ABB RobotStudio station: WriteNameStation.rspag

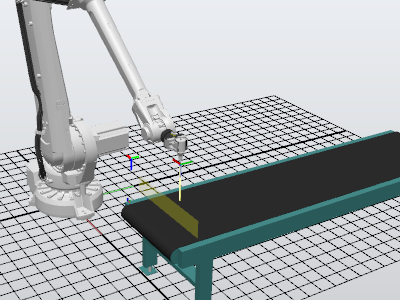
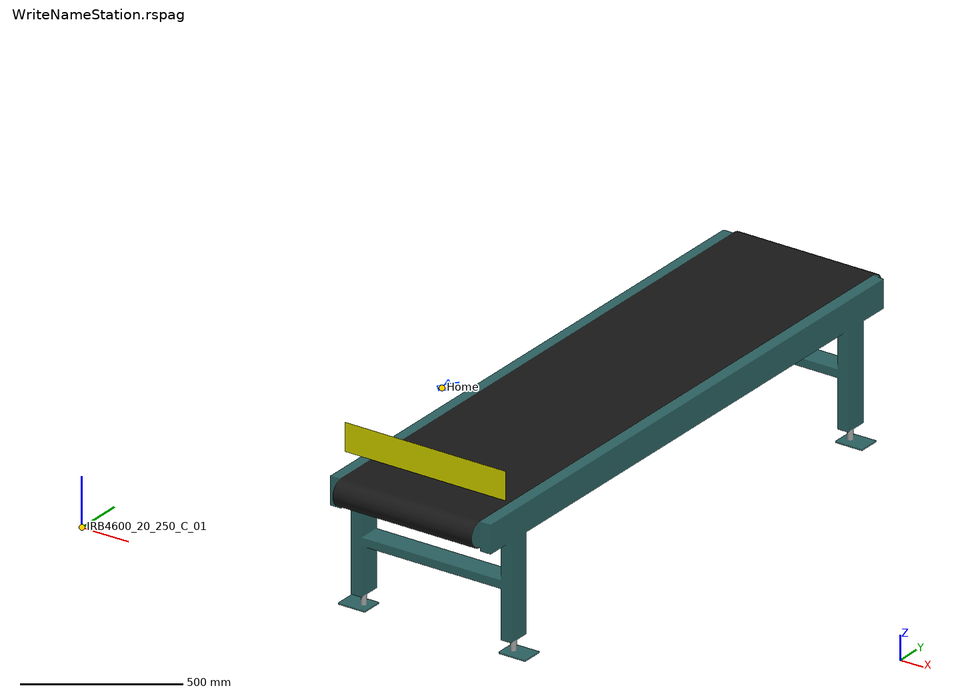
[picture v1: parts stored in the station drawn from their meshes, with robot base, taught points and paths (robot models come from the ABB library and are not in the file)]
--- station ---
Station WriteNameStation (saved by RobotStudio 23.4.10609.1)
Controller IRB4600
  mechanical unit ROB_1: IRB4600_20_250_C_01, 6 joints, base frame (0, 0, 0) mm
Layout (positions relative to the parent item):
  - IRB4600_20_250_C_01 [mechanism, from %ABB.RobotStudio.Models.IRB4600%\IRB4600_20_250_C_G_01.rslib] at (0, 0, 0) mm; joint values [0.065, -0.1396, 0.8384, 0.1009, -0.7014, -0.0772] (rad or m)
  - Belt Conveyor [part], size 703.5 x 2188.6 x 501 mm
  - Box [part], size 500 x 300 x 200 mm
  - SC_InFeeder [smart component]
      signals: DO doBoxInPos, DO doConveyorPaused, DI alwaysOn, DI diConveyor
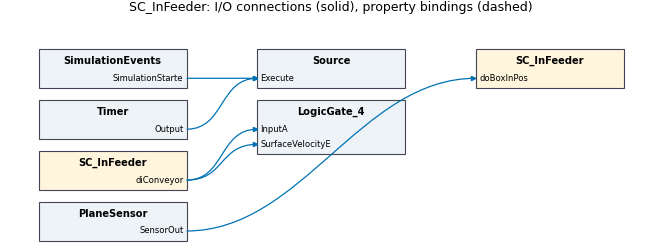
      connections:
        SimulationEvents.SimulationStarted -> Source.Execute
        Timer.Output -> Source.Execute
        SC_InFeeder.diConveyor -> LogicGate_4.InputA
        SC_InFeeder.diConveyor -> PhysicsControl.SurfaceVelocityEnabled
        PlaneSensor.SensorOut -> SC_InFeeder.doBoxInPos
    - Source [smart component, from Components\Source.rslib]
        properties: Source=Box; Copy=(none); Parent=(none); Position=[0 0 0]; Orientation=[0 0 0]; Transient=true; PhysicsBehavior=3
    - SimulationEvents [smart component, from Components\SimulationEvents.rslib]
    - Timer [smart component, from Components\Timer.rslib]
        properties: StartTime=0; Interval=5; Repeat=true; CurrentTime=12.288
    - PlaneSensor [smart component, from Components\PlaneSensor.rslib] at (984.64, 0, 535.74) mm, rotated rx 90 ry 0 rz 0 deg
        properties: Origin=[0 0 0]; Axis1=[0.6 0 0]; Axis2=[0 0.1 0]; Tag=(none); SensedPart=(none)
      - _sensorPart_ [part], size 600 x 100 x 0 mm
  - Belt [part], size 529.1 x 2200.3 x 102.1 mm
  - Pen [mechanism, from Training Objects\Pen.rslib] at (1160.02, 70, 921.71) mm, rotated rx 0 ry 90 rz 0 deg
  - SC_Painter [smart component] at (1300.02, 70, 811.71) mm, rotated rx 0 ry 0 rz -180 deg
      signals: DI diPaint
      connections:
        SC_Painter.diPaint -> PaintApplicator_4.Enabled
        LineSensor.SensedPart => PaintApplicator_4.Part
    - PaintApplicator_4 [smart component, from Components\PaintApplicator.rslib] at (0, 0, 0) mm, rotated rx 180 ry 0 rz 0 deg
        properties: Part=(none); Color=-16744256; ShowPreviewCone=true; Strength=0.6; Range=0.2; Width=0.006; Height=0.006
    - LineSensor [smart component, from Components\LineSensor.rslib] at (0, 0, 0) mm, rotated rx 180 ry 0 rz 0 deg
        properties: Start=[-2.47728111357759E-08 -5.90096643771076E-09 0.0117070722678286]; End=[-3.15805683825943E-08 -1.20119622304404E-08 0.211707072267828]; Length=0.2; Radius=0; Tag=(none); SensedPart=(none); SensedPoint=[0 0 0]
      - _sensorPart_ [part], size 0 x 0 x 200 mm
  - PhysicsControl [smart component, from Components\PhysicsControl.rslib]
      properties: Object=Belt; Behavior=2; SurfaceVelocity=0.3
Attachment: Pen is attached to IRB4600_20_250_C_01 / Link6
Attachment: PaintApplicator_4 is attached to Pen / pen
Attachment: LineSensor is attached to Pen / pen
Station logic (signal -> signal, property => property):
  SC_InFeeder.doBoxInPos -> IRB4600.diBoxInPos
  IRB4600.doPaint -> SC_Painter.diPaint
  IRB4600.doConveyor -> PhysicsControl.SurfaceVelocityEnabled
Targets, tools, work objects and paths stored in the station and not in the controller backup, written as RAPID:
! task T_ROB1
MODULE Module1
  CONST robtarget Confirmed:=[[-104.044352453,80,203.883134],[-0.000000001,0,1,0],[0,0,0,0],[9E+09,9E+09,9E+09,9E+09,9E+09,9E+09]];
  PROC Path_10()
    MoveL Home,v300,fine,Pen_TCP\WObj:=wobjInFeeder;
  ENDPROC
  PROC Path_W()
    MoveL Home,v300,fine,Pen_TCP\WObj:=wobjInFeeder;
    MoveL Offs(Home,70,0,0),v300,fine,Pen_TCP\WObj:=wobjInFeeder;
    MoveL Offs(Home,70,60,0),v300,fine,Pen_TCP\WObj:=wobjInFeeder;
    MoveL Offs(Home,85,30,0),v300,fine,Pen_TCP\WObj:=wobjInFeeder;
    MoveL Offs(Home,100,60,0),v300,fine,Pen_TCP\WObj:=wobjInFeeder;
    MoveL Offs(Home,115,0,0),v300,fine,Pen_TCP\WObj:=wobjInFeeder;
    MoveL Home,v300,fine,Pen_TCP\WObj:=wobjInFeeder;
  ENDPROC
  PROC Path_E()
    MoveL Home,v300,fine,Pen_TCP\WObj:=wobjInFeeder;
    MoveL Offs(Home,140,0,0),v300,fine,Pen_TCP\WObj:=wobjInFeeder;
    MoveL Offs(Home,140,60,0),v300,fine,Pen_TCP\WObj:=wobjInFeeder;
    MoveL Offs(Home,180,60,0),v300,fine,Pen_TCP\WObj:=wobjInFeeder;
    MoveL Offs(Home,140,30,0),v300,fine,Pen_TCP\WObj:=wobjInFeeder;
    MoveL Offs(Home,170,30,0),v300,fine,Pen_TCP\WObj:=wobjInFeeder;
    MoveL Offs(Home,140,0,0),v300,fine,Pen_TCP\WObj:=wobjInFeeder;
    MoveL Offs(Home,180,0,0),v300,fine,Pen_TCP\WObj:=wobjInFeeder;
    MoveL Home,v300,fine,Pen_TCP\WObj:=wobjInFeeder;
  ENDPROC
ENDMODULE


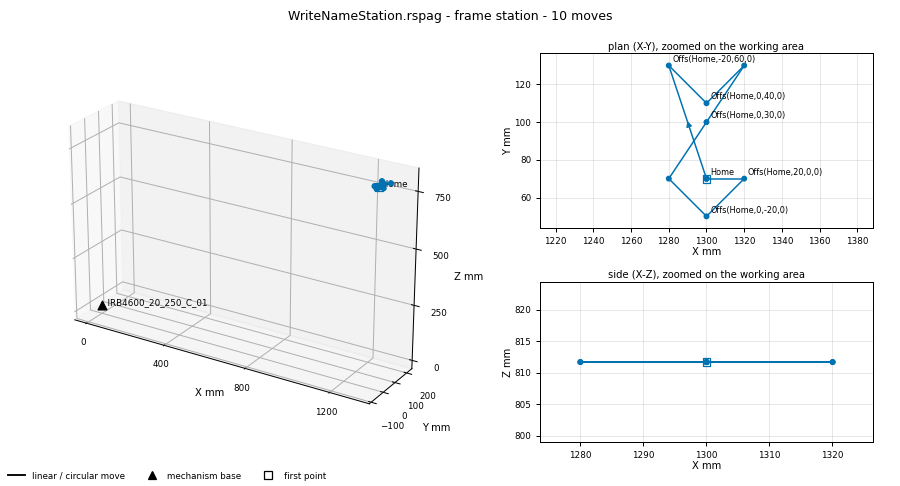
[picture p0: tool path of WriteNameStation.rspag in frame station, 10 of 10 moves have a stored position in this frame; points joined in program order, loops and branches not executed]
--- Backups/IRB4600/RAPID/TASK1/PROGMOD/CalibData.mod ---
MODULE CalibData
	PERS tooldata tVacuum:=[TRUE,[[0,0,150],[1,0,0,0]],[9,[0,0,100],[1,0,0,0],0,0,0]];
	TASK PERS wobjdata wobjInFeeder:=[FALSE,TRUE,"",[[0,0,0],[1,0,0,0]],[[1000,-80,497],[1,0,0,0]]];
    PERS tooldata Pen_TCP:=[TRUE,[[110,0,140],[0.707106781,0,0.707106781,0]],[1,[10.7435139,0,140],[1,0,0,0],0,0,0]];
ENDMODULE

--- Backups/IRB4600/RAPID/TASK1/PROGMOD/Module1.mod ---
MODULE Module1
    CONST robtarget Home:=[[300.022993432,150.000002947,314.707147681],[0.000000011,0,1,0],[0,0,-1,1],[9E+09,9E+09,9E+09,9E+09,9E+09,9E+09]];
    !***********************************************************
    !
    ! Module:  Module1
    !
    ! Description:
    !   <Insert description here>
    !
    ! Author: ander
    !
    ! Version: 1.0
    !
    !***********************************************************


    !***********************************************************
    !
    ! Procedure main
    !
    !   Smart Component example, Pick and Place application.

    !
    !***********************************************************
    PROC main()

        WHILE TRUE DO
            SetDO doConveyor, 1;

            WaitDI diBoxInPos,1;
            Path_S;

            !WaitDI diConveyorPaused,1;
            ! Confirm that the stop signal has been applied in the smart component

            !SetDO doConveyor,1;
            ! Re-enable Conveyor movement

        ENDWHILE
    ENDPROC



    PROC Path_S()
        SetDO doConveyor,0;
        ! Pause Conveyor

        MoveL Home,v300,fine,Pen_TCP\WObj:=wobjInFeeder;
        ! Move back to the Draw position or to a safe position

        SetDO doPaint,1;
        ! Enable Paint Applicator

        ! Move to the starting point of 'S'
        MoveL Offs(Home,0,0,0),v300,fine,Pen_TCP\WObj:=wobjInFeeder;
        ! Adjust the offsets as needed to position the start of 'S'

        ! Top part of 'S'
        MoveL Offs(Home,-20,60,0),v300,fine,Pen_TCP\WObj:=wobjInFeeder;
        ! Move up and to the left to start the top curve
        MoveL Offs(Home,0,40,0),v300,fine,Pen_TCP\WObj:=wobjInFeeder;
        ! Move down and to the right, continuing the top curve
        MoveL Offs(Home,20,60,0),v300,fine,Pen_TCP\WObj:=wobjInFeeder;
        ! Move up and to the right to finish the top curve

        ! Middle transition
        MoveL Offs(Home,0,30,0),v300,fine,Pen_TCP\WObj:=wobjInFeeder;
        ! Move down to start the middle part of 'S'

        ! Bottom part of 'S'
        MoveL Offs(Home,-20,0,0),v300,fine,Pen_TCP\WObj:=wobjInFeeder;
        ! Move down and to the left to start the bottom curve
        MoveL Offs(Home,0,-20,0),v300,fine,Pen_TCP\WObj:=wobjInFeeder;
        ! Move up and to the right, continuing the bottom curve
        MoveL Offs(Home,20,0,0),v300,fine,Pen_TCP\WObj:=wobjInFeeder;
        ! Move down and to the right to finish the bottom curve

        SetDO doPaint,0;

        ! Return to the draw position or to a safe position before drawing the next letter
        MoveL Home,v300,fine,Pen_TCP\WObj:=wobjInFeeder;
        ! Move back to the Draw position or to a safe position

        WaitRob\InPos;
    ENDPROC



ENDMODULE

--- Backups/IRB4600/SYSPAR/EIO.cfg ---
EIO:CFG_1.0:6:1::
#
EIO_SIGNAL:

      -Name "diBoxInPos" -SignalType "DI" -Access "All"

      -Name "doConveyor" -SignalType "DO" -Access "All" -Default 1

      -Name "diConveyorPaused" -SignalType "DI" -Access "All"

      -Name "doPaint" -SignalType "DO" -Access "All"
